Omron CX-Programmer project NewProject (CX-Programmer 9.81)

# PLC NewPLC1: CJ1M CPU11

## Program NewProgram1 (cyclic task 0)
Local symbols
Int_1 0.00 BOOL  ; int 1
Int_2 0.01 BOOL  ; Int 2
Lâmpada_1 0.02 BOOL  ; l1
Lâmpada_2 0.03 BOOL  ; l2
Lâmpada_3 0.04 BOOL  ; l3
Lâmpada_4 0.05 BOOL  ; l4

### Section MAIN

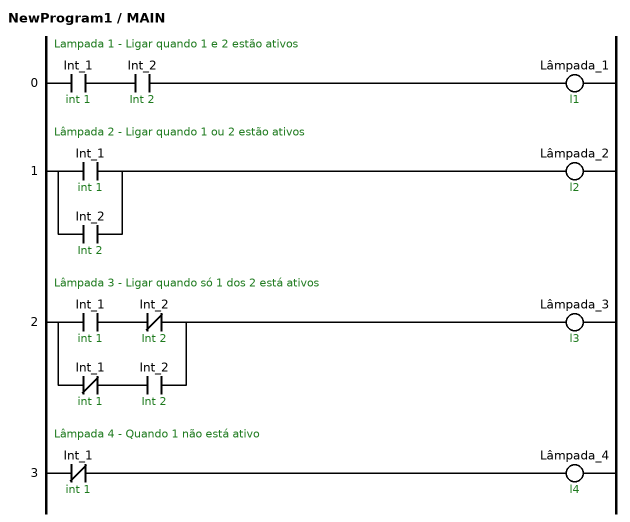
; rung 0: Lampada 1 - Ligar quando 1 e 2 estão ativos
LD Int_1  ; int 1
AND Int_2  ; Int 2
OUT Lâmpada_1  ; l1
; rung 1: Lâmpada 2 - Ligar quando 1 ou 2 estão ativos
LD Int_1  ; int 1
OR Int_2  ; Int 2
OUT Lâmpada_2  ; l2
; rung 2: Lâmpada 3 - Ligar quando só 1 dos 2 está ativos
LD Int_1  ; int 1
ANDNOT Int_2  ; Int 2
LDNOT Int_1  ; int 1
AND Int_2  ; Int 2
ORLD
OUT Lâmpada_3  ; l3
; rung 3: Lâmpada 4 - Quando 1 não está ativo
LDNOT Int_1  ; int 1
OUT Lâmpada_4  ; l4

### Section END
; rung 0
END(001)